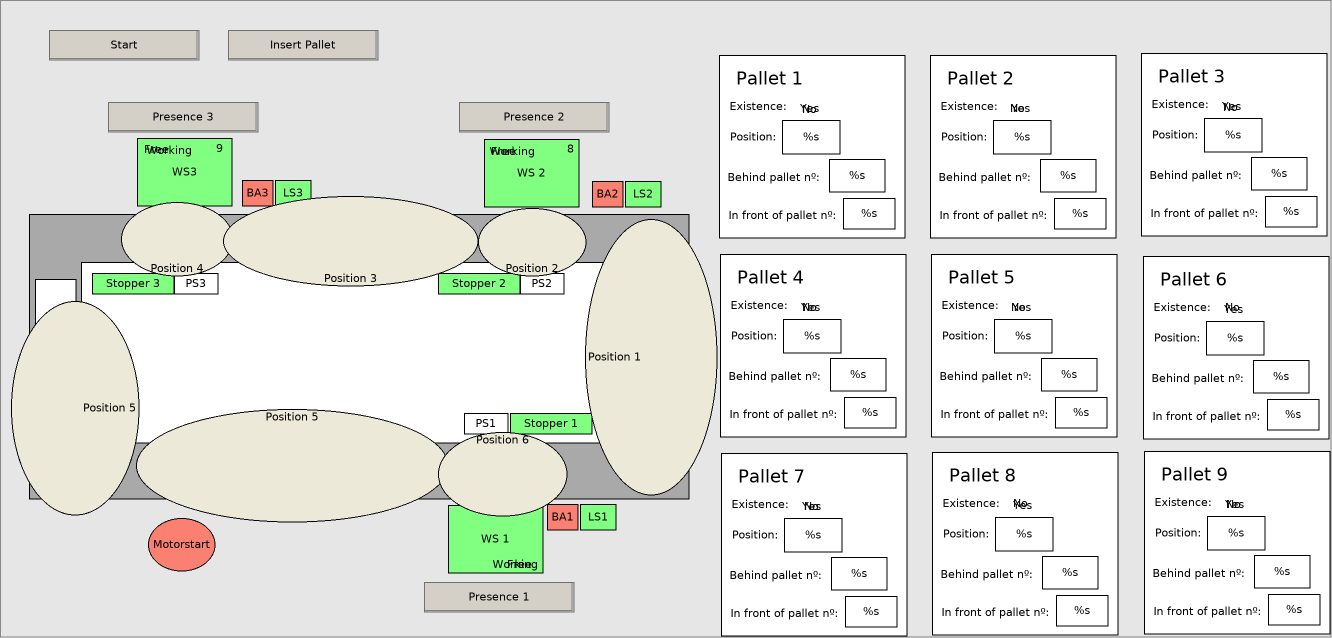
VISUALIZATION Visualization  // 1332x638
    Group (712,55 193x183)
        Rectangle (7,0 186x183)
        Label (14,0 87x47), "Pallet 1"
        Label (0,36 92x31), "Existence:"
        Label (3,65 76x34), "Position:"
        Label (3,111 117x23), "Behind pallet nº:"
        Label (12,147 117x27), "In front of pallet nº:"
        Label (64,34 67x39), "Yes", invisible if: NOT (MAIN.PALLETS[MAIN.INDEX_PALLET[1]].EX)
        Label (64,35 67x39), "No", invisible if: (MAIN.PALLETS[MAIN.INDEX_PALLET[1]].EX)
        Rectangle (70,65 58x34), "%s", text variable: MAIN.PALLETS[MAIN.INDEX_PALLET[1]].POSITION+1
        Rectangle (117,104 56x33), "%s", text variable: MAIN.PALLETS[MAIN.PALLETS[MAIN.INDEX_PALLET[1]].PREVIOUS_PALLET].NUMBER
        Rectangle (131,143 52x31), "%s", text variable: MAIN.PALLETS[MAIN.PALLETS[MAIN.INDEX_PALLET[1]].NEXT_PALLET].NUMBER
    Group (713,254 193x183)
        Rectangle (7,0 186x183)
        Label (14,0 87x47), "Pallet 4"
        Label (0,36 92x31), "Existence:"
        Label (3,65 76x34), "Position:"
        Label (3,111 117x23), "Behind pallet nº:"
        Label (12,147 117x27), "In front of pallet nº:"
        Label (64,34 67x39), "Yes", invisible if: NOT (MAIN.PALLETS[MAIN.INDEX_PALLET[4]].EX)
        Label (63,34 67x39), "No", invisible if: (MAIN.PALLETS[MAIN.INDEX_PALLET[4]].EX)
        Rectangle (70,65 58x34), "%s", text variable: MAIN.PALLETS[MAIN.INDEX_PALLET[4]].POSITION+1
        Rectangle (117,104 56x33), "%s", text variable: MAIN.PALLETS[MAIN.PALLETS[MAIN.INDEX_PALLET[4]].PREVIOUS_PALLET].NUMBER
        Rectangle (131,143 52x31), "%s", text variable: MAIN.PALLETS[MAIN.PALLETS[MAIN.INDEX_PALLET[4]].NEXT_PALLET].NUMBER
    Group (714,453 193x183)
        Rectangle (7,0 186x183)
        Label (14,0 87x47), "Pallet 7"
        Label (0,36 92x31), "Existence:"
        Label (3,65 76x34), "Position:"
        Label (3,111 117x23), "Behind pallet nº:"
        Label (12,147 117x27), "In front of pallet nº:"
        Label (64,34 67x39), "Yes", invisible if: NOT (MAIN.PALLETS[MAIN.INDEX_PALLET[7]].EX)
        Label (64,34 67x39), "No", invisible if: (MAIN.PALLETS[MAIN.INDEX_PALLET[7]].EX)
        Rectangle (70,65 58x34), "%s", text variable: MAIN.PALLETS[MAIN.INDEX_PALLET[7]].POSITION+1
        Rectangle (117,104 56x33), "%s", text variable: MAIN.PALLETS[MAIN.PALLETS[MAIN.INDEX_PALLET[7]].PREVIOUS_PALLET].NUMBER
        Rectangle (131,143 52x31), "%s", text variable: MAIN.PALLETS[MAIN.PALLETS[MAIN.INDEX_PALLET[7]].NEXT_PALLET].NUMBER
    Group (923,55 193x183)
        Rectangle (7,0 186x183)
        Label (14,0 87x47), "Pallet 2"
        Label (0,36 92x31), "Existence:"
        Label (3,65 76x34), "Position:"
        Label (3,111 117x23), "Behind pallet nº:"
        Label (12,147 117x27), "In front of pallet nº:"
        Label (64,34 67x39), "Yes", invisible if: NOT (MAIN.PALLETS[MAIN.INDEX_PALLET[2]].EX)
        Label (61,34 67x39), "No", invisible if: (MAIN.PALLETS[MAIN.INDEX_PALLET[2]].EX)
        Rectangle (70,65 58x34), "%s", text variable: MAIN.PALLETS[MAIN.INDEX_PALLET[2]].POSITION+1
        Rectangle (117,104 56x33), "%s", text variable: MAIN.PALLETS[MAIN.PALLETS[MAIN.INDEX_PALLET[2]].PREVIOUS_PALLET].NUMBER
        Rectangle (131,143 52x31), "%s", text variable: MAIN.PALLETS[MAIN.PALLETS[MAIN.INDEX_PALLET[2]].NEXT_PALLET].NUMBER
    Group (924,254 193x183)
        Rectangle (7,0 186x183)
        Label (14,0 87x47), "Pallet 5"
        Label (0,36 92x31), "Existence:"
        Label (3,65 76x34), "Position:"
        Label (3,111 117x23), "Behind pallet nº:"
        Label (12,147 117x27), "In front of pallet nº:"
        Label (64,34 67x39), "Yes", invisible if: NOT (MAIN.PALLETS[MAIN.INDEX_PALLET[5]].EX)
        Label (61,34 67x39), "No", invisible if: (MAIN.PALLETS[MAIN.INDEX_PALLET[5]].EX)
        Rectangle (70,65 58x34), "%s", text variable: MAIN.PALLETS[MAIN.INDEX_PALLET[5]].POSITION+1
        Rectangle (117,104 56x33), "%s", text variable: MAIN.PALLETS[MAIN.PALLETS[MAIN.INDEX_PALLET[5]].PREVIOUS_PALLET].NUMBER
        Rectangle (131,143 52x31), "%s", text variable: MAIN.PALLETS[MAIN.PALLETS[MAIN.INDEX_PALLET[5]].NEXT_PALLET].NUMBER
    Group (925,452 193x183)
        Rectangle (7,0 186x183)
        Label (14,0 87x47), "Pallet 8"
        Label (0,36 92x31), "Existence:"
        Label (3,65 76x34), "Position:"
        Label (3,111 117x23), "Behind pallet nº:"
        Label (12,147 117x27), "In front of pallet nº:"
        Label (64,34 67x39), "Yes", invisible if: NOT (MAIN.PALLETS[MAIN.INDEX_PALLET[8]].EX)
        Label (62,32 67x39), "No", invisible if: (MAIN.PALLETS[MAIN.INDEX_PALLET[8]].EX)
        Rectangle (70,65 58x34), "%s", text variable: MAIN.PALLETS[MAIN.INDEX_PALLET[8]].POSITION+1
        Rectangle (117,104 56x33), "%s", text variable: MAIN.PALLETS[MAIN.PALLETS[MAIN.INDEX_PALLET[8]].PREVIOUS_PALLET].NUMBER
        Rectangle (131,143 52x31), "%s", text variable: MAIN.PALLETS[MAIN.PALLETS[MAIN.INDEX_PALLET[8]].NEXT_PALLET].NUMBER
    Group (1134,53 193x183)
        Rectangle (7,0 186x183)
        Label (14,0 87x47), "Pallet 3"
        Label (0,36 92x31), "Existence:"
        Label (3,65 76x34), "Position:"
        Label (3,111 117x23), "Behind pallet nº:"
        Label (12,147 117x27), "In front of pallet nº:"
        Label (64,34 67x39), "Yes", invisible if: NOT (MAIN.PALLETS[MAIN.INDEX_PALLET[3]].EX)
        Label (63,35 67x39), "No", invisible if: (MAIN.PALLETS[MAIN.INDEX_PALLET[3]].EX)
        Rectangle (70,65 58x34), "%s", text variable: MAIN.PALLETS[MAIN.INDEX_PALLET[3]].POSITION+1
        Rectangle (117,104 56x33), "%s", text variable: MAIN.PALLETS[MAIN.PALLETS[MAIN.INDEX_PALLET[3]].PREVIOUS_PALLET].NUMBER
        Rectangle (131,143 52x31), "%s", text variable: MAIN.PALLETS[MAIN.PALLETS[MAIN.INDEX_PALLET[3]].NEXT_PALLET].NUMBER
    Group (1136,256 193x183)
        Rectangle (7,0 186x183)
        Label (14,0 87x47), "Pallet 6"
        Label (0,36 92x31), "Existence:"
        Label (3,65 76x34), "Position:"
        Label (3,111 117x23), "Behind pallet nº:"
        Label (12,147 117x27), "In front of pallet nº:"
        Label (64,34 67x39), "Yes", invisible if: NOT (MAIN.PALLETS[MAIN.INDEX_PALLET[6]].EX)
        Label (63,32 67x39), "No", invisible if: (MAIN.PALLETS[MAIN.INDEX_PALLET[6]].EX)
        Rectangle (70,65 58x34), "%s", text variable: MAIN.PALLETS[MAIN.INDEX_PALLET[6]].POSITION+1
        Rectangle (117,104 56x33), "%s", text variable: MAIN.PALLETS[MAIN.PALLETS[MAIN.INDEX_PALLET[6]].PREVIOUS_PALLET].NUMBER
        Rectangle (131,143 52x31), "%s", text variable: MAIN.PALLETS[MAIN.PALLETS[MAIN.INDEX_PALLET[6]].NEXT_PALLET].NUMBER
    Group (1137,451 193x183)
        Rectangle (7,0 186x183)
        Label (14,0 87x47), "Pallet 9"
        Label (0,36 92x31), "Existence:"
        Label (3,65 76x34), "Position:"
        Label (3,111 117x23), "Behind pallet nº:"
        Label (12,147 117x27), "In front of pallet nº:"
        Label (64,34 67x39), "Yes", invisible if: NOT (MAIN.PALLETS[MAIN.INDEX_PALLET[9]].EX)
        Label (63,34 67x39), "No", invisible if: (MAIN.PALLETS[MAIN.INDEX_PALLET[9]].EX)
        Rectangle (70,65 58x34), "%s", text variable: MAIN.PALLETS[MAIN.INDEX_PALLET[9]].POSITION+1
        Rectangle (117,104 56x33), "%s", text variable: MAIN.PALLETS[MAIN.PALLETS[MAIN.INDEX_PALLET[9]].PREVIOUS_PALLET].NUMBER
        Rectangle (131,143 52x31), "%s", text variable: MAIN.PALLETS[MAIN.PALLETS[MAIN.INDEX_PALLET[9]].NEXT_PALLET].NUMBER
    Group (11,30 706x582)
        Group (18,0 660x582)
            Button (20,0 150x30), "Start", colour toggle: MAIN.START
                tap MAIN.START
            Button (199,0 150x30), "Insert Pallet", colour toggle: MAIN.PALLET_IN
                toggle MAIN.PALLET_IN
            Button (395,552 150x30), "Presence 1", colour toggle: MAIN.P1
                toggle MAIN.P1
            Button (430,72 150x30), "Presence 2", colour toggle: MAIN.P2
                toggle MAIN.P2
            Button (79,72 150x30), "Presence 3", colour toggle: MAIN.P3
                toggle MAIN.P3
            RoundedRectangle (0,184 660x285)
            RoundedRectangle (52,232 550x181)
            Ellipse (119,488 67x53), "Motorstart", colour toggle: MAIN.MOTOR
                OnMouseDown: toggle 
            Rectangle (123,189 67x38), invisible if: NOT (MAIN.NUMBER_PALLETS[4]>0)
                OnMouseDown: toggle 
            Rectangle (213,150 31x26), "BA3", colour toggle: MAIN.BA3
                OnMouseDown: toggle 
            Rectangle (246,150 36x26), "LS3", colour toggle: MAIN.L3
                OnMouseDown: toggle 
            Rectangle (491,243 44x21), "PS2", colour toggle: MAIN.P2
                OnMouseDown: toggle 
            Rectangle (108,108 95x68), "WS3", colour toggle: MAIN.L3
                OnMouseDown: toggle 
            Rectangle (455,109 95x68), "WS 2", colour toggle: MAIN.L2
                OnMouseDown: toggle 
            Rectangle (419,475 95x68), "WS 1", colour toggle: MAIN.L1
                OnMouseDown: toggle 
            Rectangle (563,151 31x26), "BA2", colour toggle: MAIN.BA2
                OnMouseDown: toggle 
            Rectangle (596,151 36x26), "LS2", colour toggle: MAIN.L2
                OnMouseDown: toggle 
            Rectangle (518,474 31x26), "BA1", colour toggle: MAIN.BA1
                OnMouseDown: toggle 
            Rectangle (551,474 36x26), "LS1", colour toggle: MAIN.L1
                OnMouseDown: toggle 
            Rectangle (409,243 82x21), "Stopper 2", colour toggle: MAIN.S2
                OnMouseDown: toggle 
            Rectangle (145,243 44x21), "PS3", colour toggle: MAIN.P3
                OnMouseDown: toggle 
            Rectangle (63,243 82x21), "Stopper 3", colour toggle: MAIN.S3
                OnMouseDown: toggle 
            Rectangle (435,383 44x21), "PS1", colour toggle: MAIN.P1
                OnMouseDown: toggle 
            Rectangle (481,383 82x21), "Stopper 1", colour toggle: MAIN.S1
                OnMouseDown: toggle 
            Rectangle (471,189 67x37), invisible if: NOT (MAIN.NUMBER_PALLETS[2]>0)
                OnMouseDown: toggle 
            Rectangle (611,253 41x53), invisible if: NOT (MAIN.NUMBER_PALLETS[1]>=1)
                OnMouseDown: toggle 
            Label (457,524 59x21), "Working", invisible if: NOT MAIN.L1
            Label (454,111 59x21), "Working", invisible if: NOT MAIN.L2
            Label (111,110 59x21), "Working", invisible if: NOT MAIN.L3
            Label (461,524 59x21), "Free", invisible if: MAIN.L1
            Label (445,111 59x21), "Free", invisible if: MAIN.L2
            Label (98,109 59x21), "Free", invisible if: MAIN.L3
            Rectangle (613,315 41x53), invisible if: NOT (MAIN.NUMBER_PALLETS[1]=2)
                OnMouseDown: toggle 
            Rectangle (612,376 41x53), invisible if: NOT (MAIN.NUMBER_PALLETS[1]>2)
                OnMouseDown: toggle 
            Ellipse (630,318 6x4), invisible if: NOT (MAIN.NUMBER_PALLETS[1]>2)
            Ellipse (630,343 6x4), invisible if: NOT (MAIN.NUMBER_PALLETS[1]>2)
            Ellipse (630,357 6x4), invisible if: NOT (MAIN.NUMBER_PALLETS[1]>2)
            Ellipse (630,329 6x4), invisible if: NOT (MAIN.NUMBER_PALLETS[1]>2)
            Rectangle (434,421 67x38), invisible if: NOT (MAIN.NUMBER_PALLETS[6]>0)
                OnMouseDown: toggle 
            Rectangle (230,189 61x37), invisible if: NOT (MAIN.NUMBER_PALLETS[3]>=1)
                OnMouseDown: toggle 
            Rectangle (322,189 60x37), invisible if: NOT (MAIN.NUMBER_PALLETS[3]=2)
                OnMouseDown: toggle 
            Rectangle (370,188 62x38), invisible if: NOT (MAIN.NUMBER_PALLETS[3]>2)
                OnMouseDown: toggle 
            Ellipse (304,207 6x4), invisible if: NOT (MAIN.NUMBER_PALLETS[3]>2)
            Ellipse (325,207 6x4), invisible if: NOT (MAIN.NUMBER_PALLETS[3]>2)
            Ellipse (348,207 6x4), invisible if: NOT (MAIN.NUMBER_PALLETS[3]>2)
            Rectangle (6,249 41x53), invisible if: NOT (MAIN.NUMBER_PALLETS[5]>=1)
                OnMouseDown: toggle 
            Rectangle (6,328 41x53), invisible if: NOT (MAIN.NUMBER_PALLETS[5]=2)
                OnMouseDown: toggle 
            Rectangle (276,418 61x43), invisible if: NOT (MAIN.NUMBER_PALLETS[5]>2)
                OnMouseDown: toggle 
            Ellipse (226,435 6x4), invisible if: NOT (MAIN.NUMBER_PALLETS[5]>2)
            Ellipse (178,435 6x4), invisible if: NOT (MAIN.NUMBER_PALLETS[5]>2)
            Ellipse (127,437 6x4), invisible if: NOT (MAIN.NUMBER_PALLETS[5]>2)
            Ellipse (73,435 6x4), invisible if: NOT (MAIN.NUMBER_PALLETS[5]>2)
            Ellipse (24,393 6x4), invisible if: NOT (MAIN.NUMBER_PALLETS[5]>2)
            Ellipse (23,341 6x4), invisible if: NOT (MAIN.NUMBER_PALLETS[5]>2)
            Ellipse (449,178 108x68), "Position 2"
            Ellipse (92,172 112x74), "Position 4"
            Ellipse (107,379 312x113), "Position 5"
            Ellipse (409,402 129x84), "Position 6"
            Label (527,106 29x26), "8"
            Label (178,108 25x21), "9"
        Ellipse (574,189 132x276), "Position 1"
        Ellipse (212,166 255x90), "Position 3"
        Ellipse (0,271 128x214), "Position 5"
END_VISUALIZATION

(* stored: Version 1.1.0.1, ProductVersion 3.1.4020.6
   Visu Visualization: Id {03c63bfc-dd13-433d-b315-0d49675523c2} *)
